# EPICS substitutions: apps/scalerApp/Db/scaler-ped.substitutions
file "db/scaler-ped.db" {
pattern { P           RAW        REF      REFMAX RAWMAX WINDOW HALFWINDOW NPED OUT         VETO }
        { fcup_offset scalerS2b  IPM2C21A 0.01   -1     17     9          10   fcup_offset scaler_mode }
        { slm_offset  scalerS16b IPM2C21A 0.01   -1     17     9          10   slm_offset  scaler_mode }
}
